Universal Robots PolyScope program: back.urp

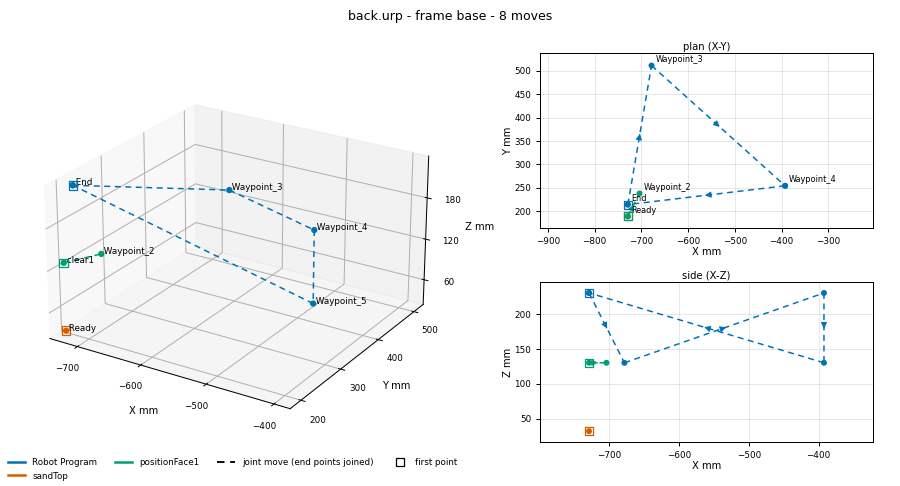
[picture p0: tool path of back.urp in frame base, 8 of 8 moves have a stored position in this frame; points joined in program order, loops and branches not executed]
Program back (installation=default directory=/programs/new folder createdIn=5.11.5.1010327 lastSavedIn=5.11.5.1010327 robotSerialNumber=20215500677)
Calibrated DH parameters: a=[0.000204, -0.239222, -0.391845, -0.000001, 0.000022, 0]; d=[0.162722, -355.808559, 353.37206, 2.570385, 0.099741, 0.099629]; alpha=[1.571124, 0.000988, 0.008295, 1.568963, -1.570303, 0]; deltaTheta=[0, -0.973091, 7.204745, 0.05153, 0, 0]
Robot Program (runOnlyOnce=true)
  Set NoAction tcp=Dynabrade1
  MoveJ speed 60 deg/s, acceleration 80 deg/s^2 (useActiveTCP=true) feature=Point_1
    Waypoint End: TCP in base x=-728.9 y=214.201 z=230.404 mm, rx=-0.0043 ry=-3.1415 rz=-0.0001 rad; joints [333.501, -52.135, 61.248, -99.09, -89.528, 243.76] deg; TCP offset x=0 y=0 z=105 mm, rx=0 ry=0 rz=0 rad; feature pose in base x=-728.914 y=214.233 z=30.379 mm, rx=0 ry=0 rz=3.1416 rad
  Call sandTop
  Call positionFace1
  Call sandFace
  MoveJ speed 60 deg/s, acceleration 80 deg/s^2 (useActiveTCP=true) feature=Point_1
    Waypoint Waypoint_3: TCP in base x=-678.243 y=511.665 z=130.309 mm, rx=-1.5708 ry=-0.0001 rz=0 rad; joints [325.381, -29.88, 51.308, -20.942, 145.47, 180.606] deg; TCP offset x=0 y=0 z=105 mm, rx=0 ry=0 rz=0 rad; feature pose in base x=-728.914 y=189 z=30.379 mm, rx=0 ry=0 rz=3.1416 rad
  Call sandFace
  MoveJ speed 60 deg/s, acceleration 80 deg/s^2 (useActiveTCP=true) feature=Point_1
    Waypoint Waypoint_4: TCP in base x=-392.425 y=254.355 z=230.384 mm, rx=1.2093 ry=1.2091 rz=1.2093 rad; joints [325.12, -49.665, 73.027, -23.568, -124.766, -0.394] deg
    Waypoint Waypoint_5: TCP in base x=-392.412 y=254.363 z=130.395 mm, rx=1.2094 ry=1.2091 rz=1.2092 rad; joints [325.114, -42.907, 77.192, -34.469, -124.689, -0.353] deg
  Call sandFace
  URCap Finishing Tool Control (Robotiq_Copilot, Robotiq Inc.) dataModel(FinishingToolStateKey=false, ToolOutputNameKey=digital_out[0], HackTriggeringContributionIsDefinedMethodKey=true)
  MoveJ speed 60 deg/s, acceleration 80 deg/s^2 (useActiveTCP=true) feature=Point_1
    Waypoint End: TCP in base x=-728.9 y=214.201 z=230.404 mm, rx=-0.0043 ry=-3.1415 rz=-0.0001 rad; joints [333.501, -52.135, 61.248, -99.09, -89.528, 243.76] deg; TCP offset x=0 y=0 z=105 mm, rx=0 ry=0 rz=0 rad; feature pose in base x=-728.914 y=214.233 z=30.379 mm, rx=0 ry=0 rz=3.1416 rad
SubProgram -> positionFace1
SubProgram -> sandFace
SubProgram -> sandTop
SubProgram sandEdges1 [hidden by the author, left out]
SubProgram sandTop (keepSynchronizedWithDisk=true) programFile=/programs/new folder/sandTop.urp
  MoveJ speed 60 deg/s, acceleration 80 deg/s^2 (useActiveTCP=false) tcp=Dynabrade1; feature=Point_1
    Waypoint Ready: TCP in base x=-728.914 y=189 z=32.379 mm, rx=0 ry=-3.1416 rz=0 rad; joints [335.226, -42.704, 75.581, -122.851, -89.577, 245.512] deg; TCP offset x=0 y=0 z=105 mm, rx=0 ry=0 rz=0 rad; feature pose in base x=-728.914 y=189 z=30.379 mm, rx=0 ry=0 rz=3.1416 rad
  MoveL speed 250 mm/s, acceleration 1200 mm/s^2 (useActiveTCP=true) feature=Base
    MoveDirectionNode (selectedDirection=ZMinus)
      Until TOOL_CONTACT_DETECTION (allowActions=false retraction=0 decelerationAcceleration=3 decelerationAngularAcceleration=34.906585)
  URCap Finishing Tool Control (Robotiq_Copilot, Robotiq Inc.) dataModel(ToolOutputNameKey=digital_out[0], HackTriggeringContributionIsDefinedMethodKey=true)
  Wait Sleep waitTime=0.5
  Force Simple feature=Joint_6_name; selection=[0, 0, 1, 0, 0, 0]; wrench=[0, 0, 3, 0, 0, 0]; limitsForce=[0.15, 0.15, 0.15, 1.047198, 1.047198, 1.047198]; limitsMotion=[0.1, 0.1, 0.1, 0.349066, 0.349066, 0.349066]
    SuppressedNode
      MoveL speed 60 mm/s, acceleration 1200 mm/s^2 (useActiveTCP=true) feature=CubeTop
        Waypoint corner1: TCP in base x=-728.953 y=214.204 z=30.412 mm, rx=0.0002 ry=-3.1414 rz=-0.0001 rad; joints [333.479, -41.753, 74.065, -122.295, -89.572, 243.755] deg; TCP offset x=0 y=0 z=105 mm, rx=0 ry=0 rz=0 rad; feature pose in base x=-763.485 y=236.346 z=30.378 mm, rx=0.0002 ry=-0.0001 rz=0.0002 rad
        Waypoint corner2: TCP in base x=-557.584 y=356.051 z=312.282 mm, rx=1.2185 ry=2.8111 rz=0.1357 rad; joints [317.739, -66.413, 71.003, -92.128, -95.717, 274.795] deg; feature pose in base x=-763.485 y=236.346 z=30.378 mm, rx=0.0002 ry=-0.0001 rz=0.0002 rad
        Waypoint corner3: TCP in base x=-331.315 y=581.729 z=28.44 mm, rx=-0.7341 ry=-3.0546 rz=-0.0003 rad; joints [288.115, -51.53, 93.339, -131.791, -89.632, 225.49] deg; TCP offset x=0 y=0 z=105 mm, rx=0 ry=0 rz=0 rad; feature pose in base x=-765.472 y=232.505 z=32.467 mm, rx=0.4889 ry=-3.103 rz=-0.001 rad
        Waypoint corner4: TCP in base x=-331.396 y=226.729 z=28.426 mm, rx=-0.7341 ry=-3.0545 rz=0 rad; joints [306.044, -77.589, 138.917, -151.305, -89.768, 243.54] deg; TCP offset x=0 y=0 z=105 mm, rx=0 ry=0 rz=0 rad
        Waypoint corner1: TCP in base x=-728.953 y=214.204 z=30.412 mm, rx=0.0002 ry=-3.1414 rz=-0.0001 rad; joints [333.479, -41.753, 74.065, -122.295, -89.572, 243.755] deg; TCP offset x=0 y=0 z=105 mm, rx=0 ry=0 rz=0 rad; feature pose in base x=-763.485 y=236.346 z=30.378 mm, rx=0.0002 ry=-0.0001 rz=0.0002 rad
    MoveL speed 30 mm/s, acceleration 1200 mm/s^2 (useActiveTCP=true) feature=Base
      MoveDirectionNode (selectedDirection=YPlus)
        Until DISTANCE (allowActions=false deceleration=3 distanceNodeType=BLEND) Distance=0.35; motionParameters(blendRadius=0.005)
      MoveDirectionNode (selectedDirection=XPlus)
        Until DISTANCE (allowActions=false deceleration=3 distanceNodeType=BLEND) Distance=0.36; motionParameters(blendRadius=0.005)
      MoveDirectionNode (selectedDirection=YMinus)
        Until DISTANCE (allowActions=false deceleration=3 distanceNodeType=BLEND) Distance=0.35; motionParameters(blendRadius=0.005)
      MoveDirectionNode (selectedDirection=XMinus)
        Until DISTANCE (allowActions=false deceleration=3 distanceNodeType=STOP) Distance=0.36; motionParameters(blendRadius=0.005)
  MoveL speed 60 mm/s, acceleration 1200 mm/s^2 (useActiveTCP=true) feature=Base
    MoveDirectionNode (selectedDirection=ZPlus)
      Until DISTANCE (allowActions=false deceleration=3 distanceNodeType=STOP) Distance=0.025; motionParameters(blendRadius=0)
  URCap Finishing Tool Control (Robotiq_Copilot, Robotiq Inc.) dataModel(ToolOutputNameKey=digital_out[0], HackTriggeringContributionIsDefinedMethodKey=true, FinishingToolStateKey=false)
SubProgram positionFace1 (keepSynchronizedWithDisk=false) programFile=/programs/new folder/faces1.urp
  MoveJ speed 60 deg/s, acceleration 80 deg/s^2 (useActiveTCP=true) feature=Point_1
    Waypoint clear1: TCP in base x=-728.908 y=189.012 z=130.386 mm, rx=0 ry=-3.1416 rz=0 rad; joints [335.235, -49.1, 71.247, -112.122, -89.547, 245.44] deg; feature pose in base x=-728.914 y=189 z=30.379 mm, rx=0 ry=0 rz=3.1416 rad
    Waypoint Waypoint_2: TCP in base x=-703.919 y=237.998 z=130.399 mm, rx=-1.2091 ry=-1.2091 rz=1.2092 rad; joints [320.596, -53.202, 97.124, -44.178, 50.855, 180.356] deg
SubProgram sandFace (keepSynchronizedWithDisk=false)
  MoveL speed 30 mm/s, acceleration 1200 mm/s^2 (useActiveTCP=true) feature=Base
    MoveDirectionNode (selectedDirection=ZMinus)
      Until DISTANCE (allowActions=false deceleration=3 distanceNodeType=STOP) Distance=0.046; motionParameters(blendRadius=0)
    MoveDirectionNode (selectedDirection=ZPlus) feature=Joint_6_name
      Until TOOL_CONTACT_DETECTION (allowActions=false retraction=0 decelerationAcceleration=3 decelerationAngularAcceleration=34.906585)
    URCap Finishing Tool Control (Robotiq_Copilot, Robotiq Inc.) dataModel(ToolOutputNameKey=digital_out[0], HackTriggeringContributionIsDefinedMethodKey=true)
    Force Simple feature=Joint_6_name; selection=[0, 0, 1, 0, 0, 0]; wrench=[0, 0, 5, 0, 0, 0]; limitsForce=[0.15, 0.15, 0.15, 1.047198, 1.047198, 1.047198]; limitsMotion=[0.1, 0.1, 0.1, 0.349066, 0.349066, 0.349066]
      MoveDirectionNode (selectedDirection=XPlus) feature=Joint_6_name
        Until DISTANCE (allowActions=false deceleration=3 distanceNodeType=STOP) Distance=0.26; motionParameters(blendRadius=0)
    URCap Finishing Tool Control (Robotiq_Copilot, Robotiq Inc.) dataModel(FinishingToolStateKey=false, ToolOutputNameKey=digital_out[0], HackTriggeringContributionIsDefinedMethodKey=true)
    MoveDirectionNode (selectedDirection=ZPlus)
      Until DISTANCE (allowActions=false deceleration=3 distanceNodeType=STOP) Distance=0.05; motionParameters(blendRadius=0)
